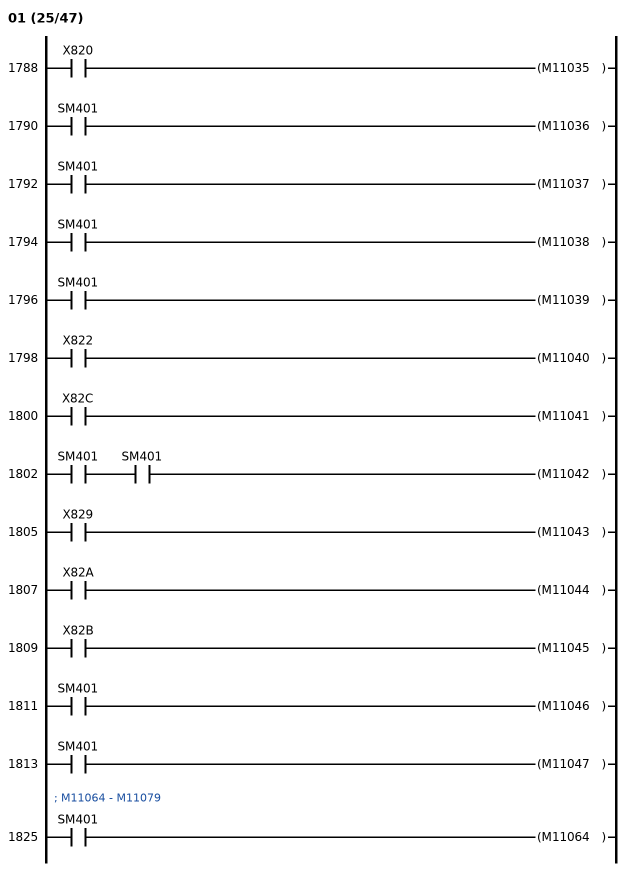
1788  LD      X820
      OUT     M11035
1790  LD      SM401
      OUT     M11036
1792  LD      SM401
      OUT     M11037
1794  LD      SM401
      OUT     M11038
1796  LD      SM401
      OUT     M11039
1798  LD      X822
      OUT     M11040
1800  LD      X82C
      OUT     M11041
1802  LD      SM401
      AND     SM401
      OUT     M11042
1805  LD      X829
      OUT     M11043
1807  LD      X82A
      OUT     M11044
1809  LD      X82B
      OUT     M11045
1811  LD      SM401
      OUT     M11046
1813  LD      SM401
      OUT     M11047
; M11064 - M11079
1825  LD      SM401
      OUT     M11064
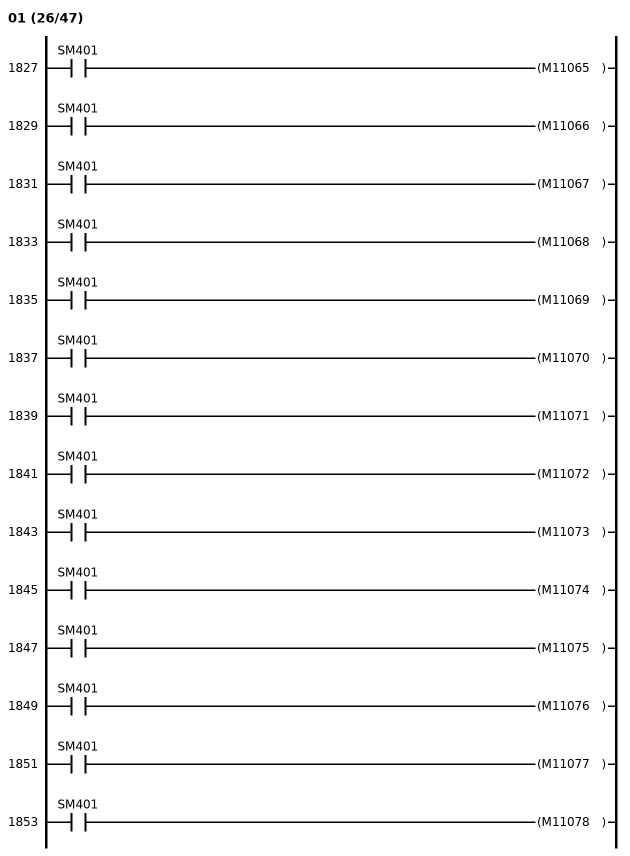
1827  LD      SM401
      OUT     M11065
1829  LD      SM401
      OUT     M11066
1831  LD      SM401
      OUT     M11067
1833  LD      SM401
      OUT     M11068
1835  LD      SM401
      OUT     M11069
1837  LD      SM401
      OUT     M11070
1839  LD      SM401
      OUT     M11071
1841  LD      SM401
      OUT     M11072
1843  LD      SM401
      OUT     M11073
1845  LD      SM401
      OUT     M11074
1847  LD      SM401
      OUT     M11075
1849  LD      SM401
      OUT     M11076
1851  LD      SM401
      OUT     M11077
1853  LD      SM401
      OUT     M11078
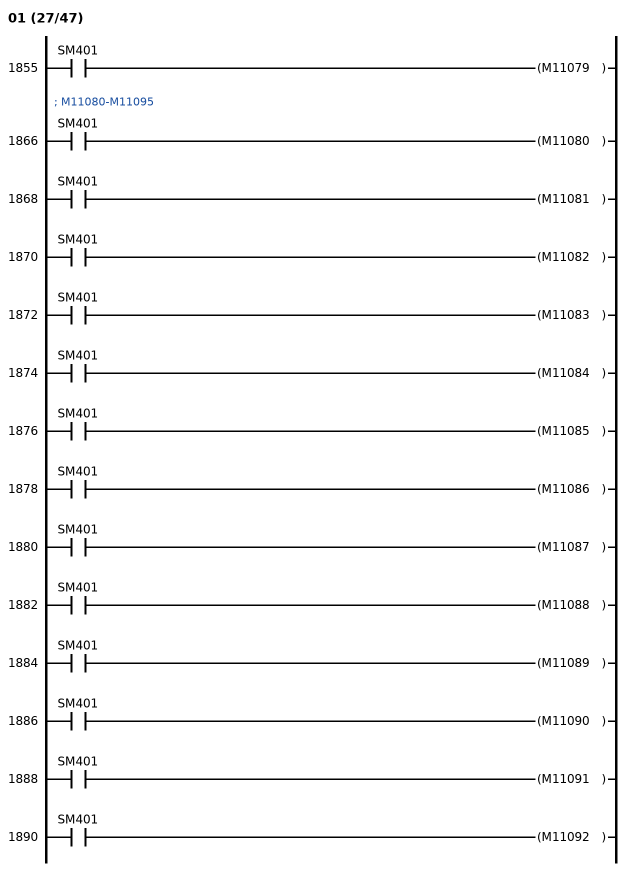
1855  LD      SM401
      OUT     M11079
; M11080-M11095
1866  LD      SM401
      OUT     M11080
1868  LD      SM401
      OUT     M11081
1870  LD      SM401
      OUT     M11082
1872  LD      SM401
      OUT     M11083
1874  LD      SM401
      OUT     M11084
1876  LD      SM401
      OUT     M11085
1878  LD      SM401
      OUT     M11086
1880  LD      SM401
      OUT     M11087
1882  LD      SM401
      OUT     M11088
1884  LD      SM401
      OUT     M11089
1886  LD      SM401
      OUT     M11090
1888  LD      SM401
      OUT     M11091
1890  LD      SM401
      OUT     M11092
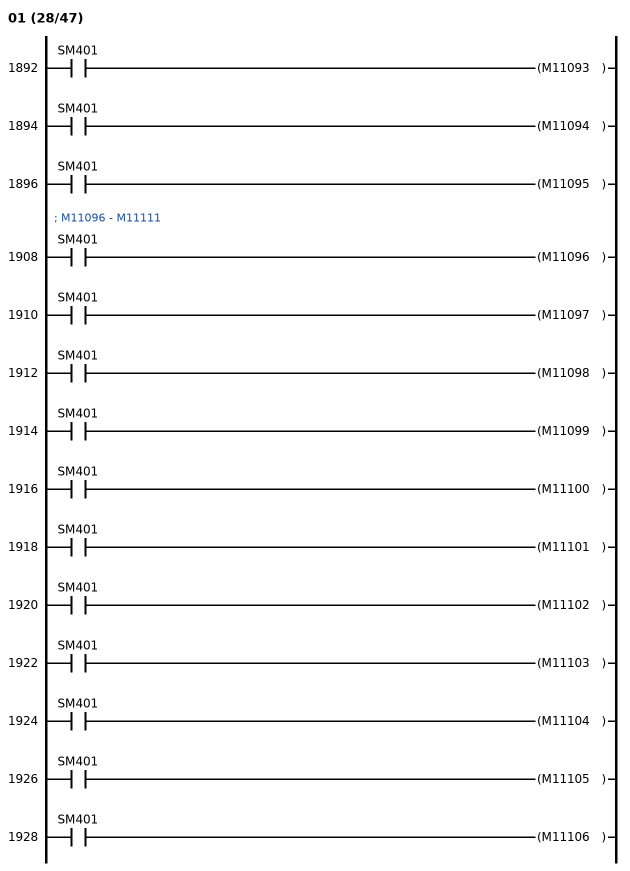
1892  LD      SM401
      OUT     M11093
1894  LD      SM401
      OUT     M11094
1896  LD      SM401
      OUT     M11095
; M11096 - M11111
1908  LD      SM401
      OUT     M11096
1910  LD      SM401
      OUT     M11097
1912  LD      SM401
      OUT     M11098
1914  LD      SM401
      OUT     M11099
1916  LD      SM401
      OUT     M11100
1918  LD      SM401
      OUT     M11101
1920  LD      SM401
      OUT     M11102
1922  LD      SM401
      OUT     M11103
1924  LD      SM401
      OUT     M11104
1926  LD      SM401
      OUT     M11105
1928  LD      SM401
      OUT     M11106
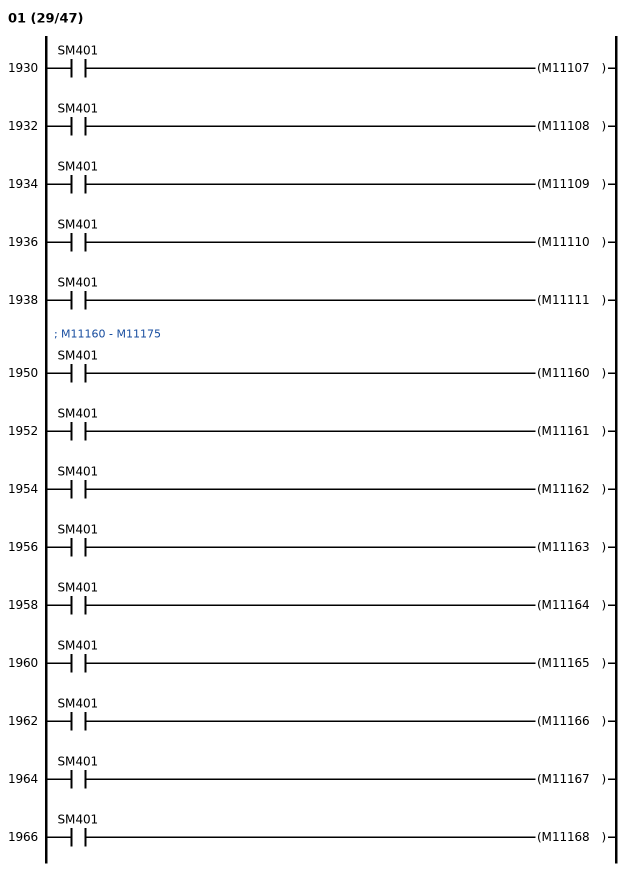
1930  LD      SM401
      OUT     M11107
1932  LD      SM401
      OUT     M11108
1934  LD      SM401
      OUT     M11109
1936  LD      SM401
      OUT     M11110
1938  LD      SM401
      OUT     M11111
; M11160 - M11175
1950  LD      SM401
      OUT     M11160
1952  LD      SM401
      OUT     M11161
1954  LD      SM401
      OUT     M11162
1956  LD      SM401
      OUT     M11163
1958  LD      SM401
      OUT     M11164
1960  LD      SM401
      OUT     M11165
1962  LD      SM401
      OUT     M11166
1964  LD      SM401
      OUT     M11167
1966  LD      SM401
      OUT     M11168
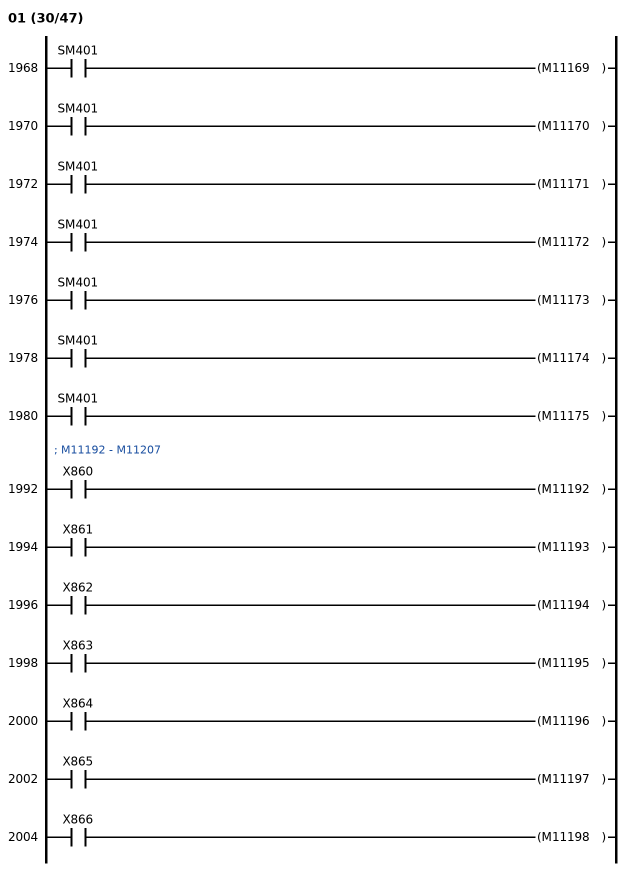
1968  LD      SM401
      OUT     M11169
1970  LD      SM401
      OUT     M11170
1972  LD      SM401
      OUT     M11171
1974  LD      SM401
      OUT     M11172
1976  LD      SM401
      OUT     M11173
1978  LD      SM401
      OUT     M11174
1980  LD      SM401
      OUT     M11175
; M11192 - M11207
1992  LD      X860
      OUT     M11192
1994  LD      X861
      OUT     M11193
1996  LD      X862
      OUT     M11194
1998  LD      X863
      OUT     M11195
2000  LD      X864
      OUT     M11196
2002  LD      X865
      OUT     M11197
2004  LD      X866
      OUT     M11198
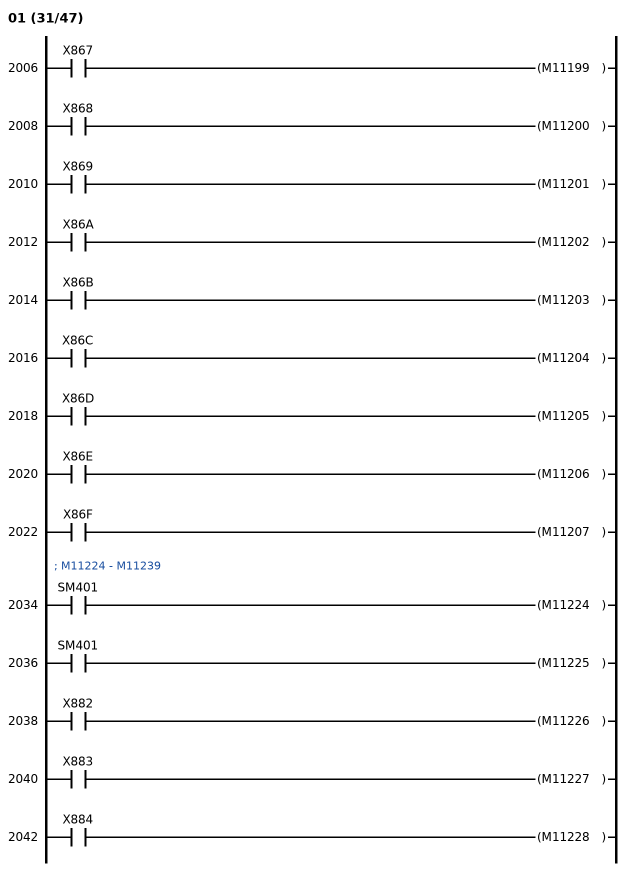
2006  LD      X867
      OUT     M11199
2008  LD      X868
      OUT     M11200
2010  LD      X869
      OUT     M11201
2012  LD      X86A
      OUT     M11202
2014  LD      X86B
      OUT     M11203
2016  LD      X86C
      OUT     M11204
2018  LD      X86D
      OUT     M11205
2020  LD      X86E
      OUT     M11206
2022  LD      X86F
      OUT     M11207
; M11224 - M11239
2034  LD      SM401
      OUT     M11224
2036  LD      SM401
      OUT     M11225
2038  LD      X882
      OUT     M11226
2040  LD      X883
      OUT     M11227
2042  LD      X884
      OUT     M11228
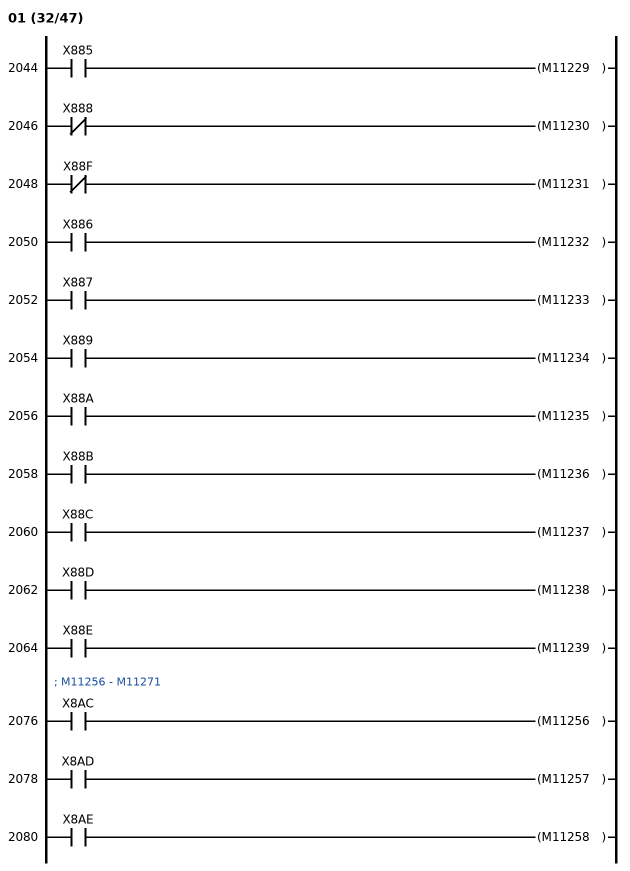
2044  LD      X885
      OUT     M11229
2046  LDI     X888
      OUT     M11230
2048  LDI     X88F
      OUT     M11231
2050  LD      X886
      OUT     M11232
2052  LD      X887
      OUT     M11233
2054  LD      X889
      OUT     M11234
2056  LD      X88A
      OUT     M11235
2058  LD      X88B
      OUT     M11236
2060  LD      X88C
      OUT     M11237
2062  LD      X88D
      OUT     M11238
2064  LD      X88E
      OUT     M11239
; M11256 - M11271
2076  LD      X8AC
      OUT     M11256
2078  LD      X8AD
      OUT     M11257
2080  LD      X8AE
      OUT     M11258
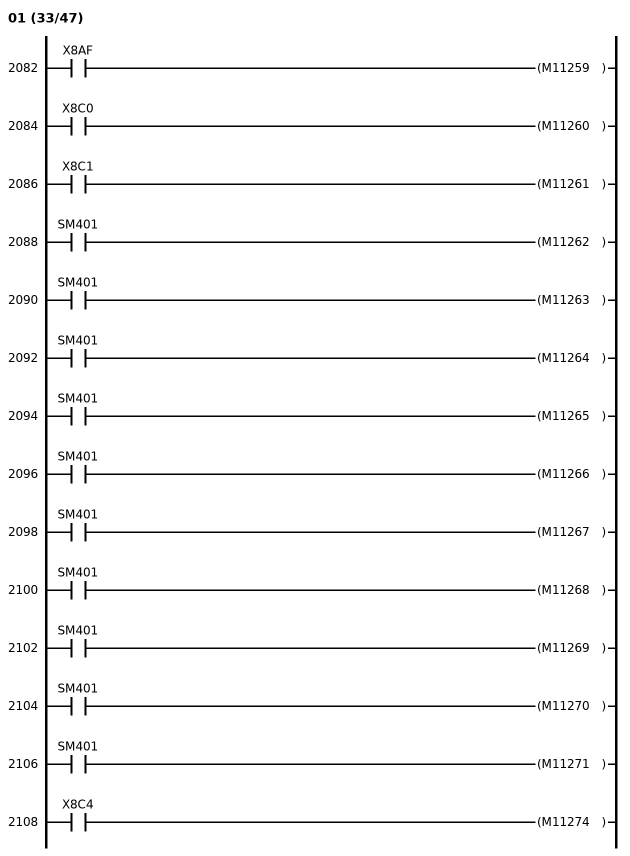
2082  LD      X8AF
      OUT     M11259
2084  LD      X8C0
      OUT     M11260
2086  LD      X8C1
      OUT     M11261
2088  LD      SM401
      OUT     M11262
2090  LD      SM401
      OUT     M11263
2092  LD      SM401
      OUT     M11264
2094  LD      SM401
      OUT     M11265
2096  LD      SM401
      OUT     M11266
2098  LD      SM401
      OUT     M11267
2100  LD      SM401
      OUT     M11268
2102  LD      SM401
      OUT     M11269
2104  LD      SM401
      OUT     M11270
2106  LD      SM401
      OUT     M11271
2108  LD      X8C4
      OUT     M11274
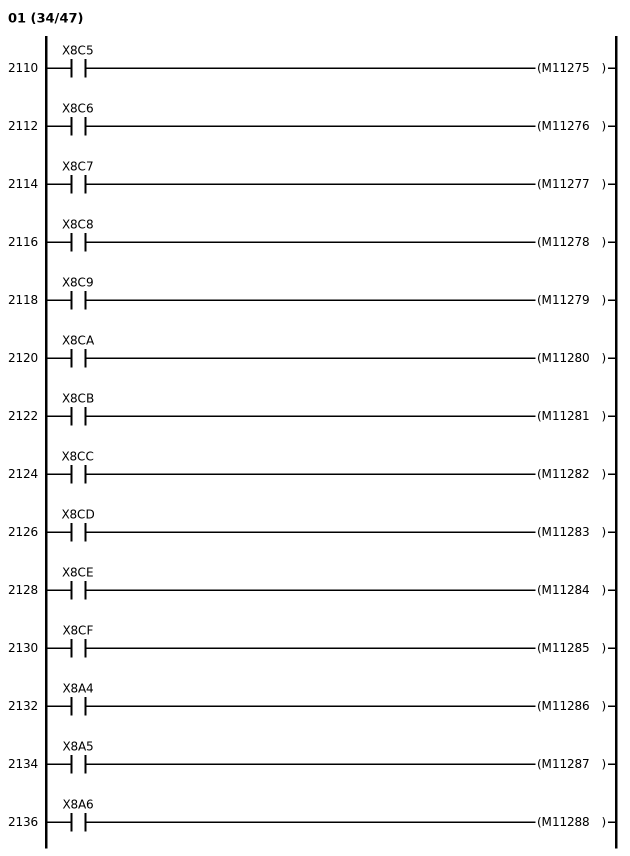
2110  LD      X8C5
      OUT     M11275
2112  LD      X8C6
      OUT     M11276
2114  LD      X8C7
      OUT     M11277
2116  LD      X8C8
      OUT     M11278
2118  LD      X8C9
      OUT     M11279
2120  LD      X8CA
      OUT     M11280
2122  LD      X8CB
      OUT     M11281
2124  LD      X8CC
      OUT     M11282
2126  LD      X8CD
      OUT     M11283
2128  LD      X8CE
      OUT     M11284
2130  LD      X8CF
      OUT     M11285
2132  LD      X8A4
      OUT     M11286
2134  LD      X8A5
      OUT     M11287
2136  LD      X8A6
      OUT     M11288
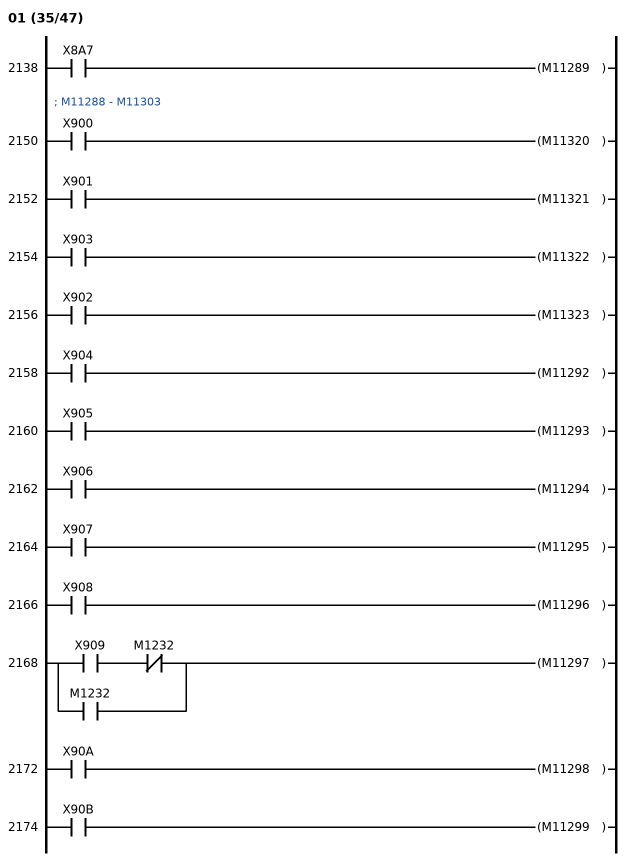
2138  LD      X8A7
      OUT     M11289
; M11288 - M11303
2150  LD      X900
      OUT     M11320
2152  LD      X901
      OUT     M11321
2154  LD      X903
      OUT     M11322
2156  LD      X902
      OUT     M11323
2158  LD      X904
      OUT     M11292
2160  LD      X905
      OUT     M11293
2162  LD      X906
      OUT     M11294
2164  LD      X907
      OUT     M11295
2166  LD      X908
      OUT     M11296
2168  LD      X909
      ANI     M1232
      OR      M1232
      OUT     M11297
2172  LD      X90A
      OUT     M11298
2174  LD      X90B
      OUT     M11299
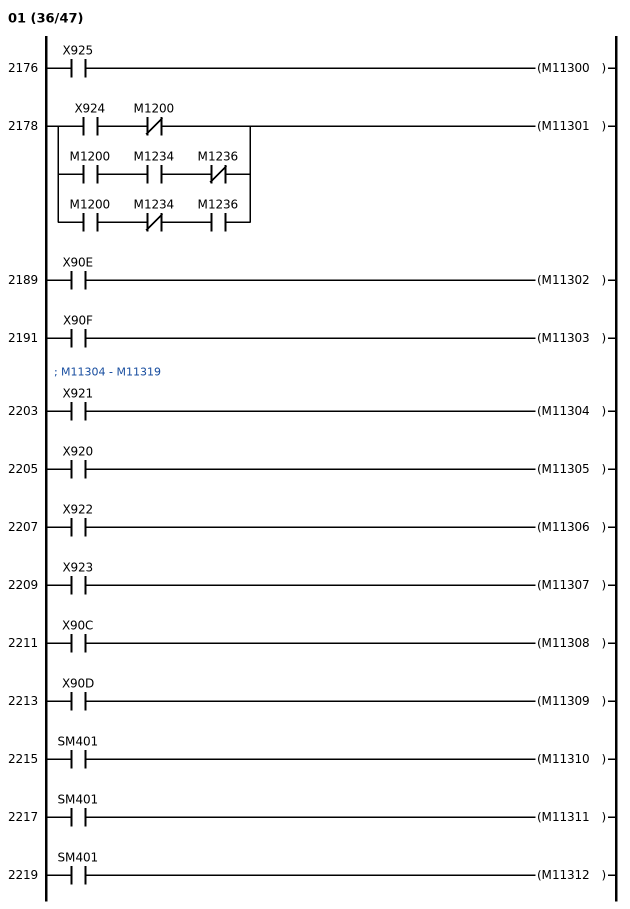
2176  LD      X925
      OUT     M11300
2178  LD      X924
      ANI     M1200
      LD      M1200
      AND     M1234
      ANI     M1236
      ORB
      LD      M1200
      ANI     M1234
      AND     M1236
      ORB
      OUT     M11301
2189  LD      X90E
      OUT     M11302
2191  LD      X90F
      OUT     M11303
; M11304 - M11319
2203  LD      X921
      OUT     M11304
2205  LD      X920
      OUT     M11305
2207  LD      X922
      OUT     M11306
2209  LD      X923
      OUT     M11307
2211  LD      X90C
      OUT     M11308
2213  LD      X90D
      OUT     M11309
2215  LD      SM401
      OUT     M11310
2217  LD      SM401
      OUT     M11311
2219  LD      SM401
      OUT     M11312
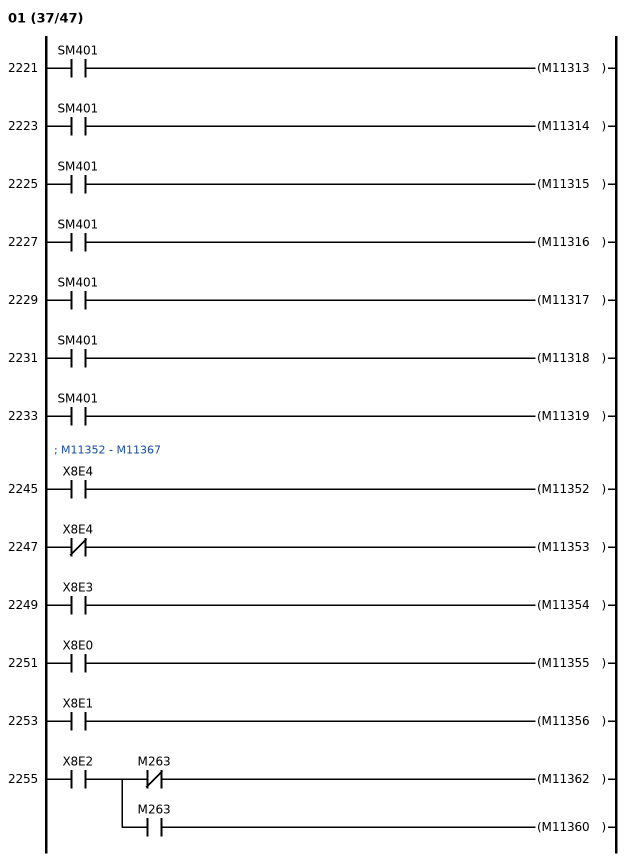
2221  LD      SM401
      OUT     M11313
2223  LD      SM401
      OUT     M11314
2225  LD      SM401
      OUT     M11315
2227  LD      SM401
      OUT     M11316
2229  LD      SM401
      OUT     M11317
2231  LD      SM401
      OUT     M11318
2233  LD      SM401
      OUT     M11319
; M11352 - M11367
2245  LD      X8E4
      OUT     M11352
2247  LDI     X8E4
      OUT     M11353
2249  LD      X8E3
      OUT     M11354
2251  LD      X8E0
      OUT     M11355
2253  LD      X8E1
      OUT     M11356
2255  LD      X8E2
      MPS
      ANI     M263
      OUT     M11362
      MPP
      AND     M263
      OUT     M11360
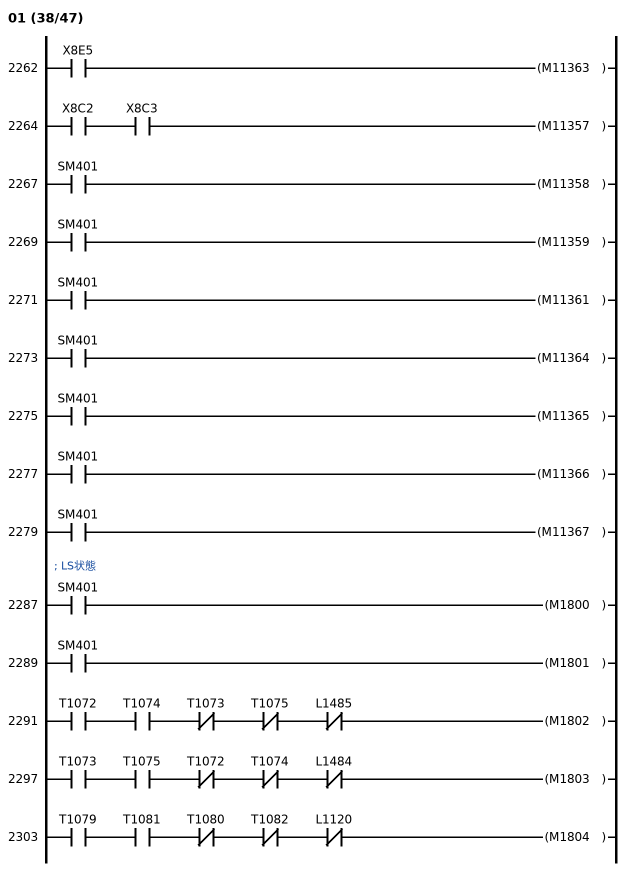
2262  LD      X8E5
      OUT     M11363
2264  LD      X8C2
      AND     X8C3
      OUT     M11357
2267  LD      SM401
      OUT     M11358
2269  LD      SM401
      OUT     M11359
2271  LD      SM401
      OUT     M11361
2273  LD      SM401
      OUT     M11364
2275  LD      SM401
      OUT     M11365
2277  LD      SM401
      OUT     M11366
2279  LD      SM401
      OUT     M11367
; LS状態
2287  LD      SM401
      OUT     M1800
2289  LD      SM401
      OUT     M1801
2291  LD      T1072
      AND     T1074
      ANI     T1073
      ANI     T1075
      ANI     L1485
      OUT     M1802
2297  LD      T1073
      AND     T1075
      ANI     T1072
      ANI     T1074
      ANI     L1484
      OUT     M1803
2303  LD      T1079
      AND     T1081
      ANI     T1080
      ANI     T1082
      ANI     L1120
      OUT     M1804
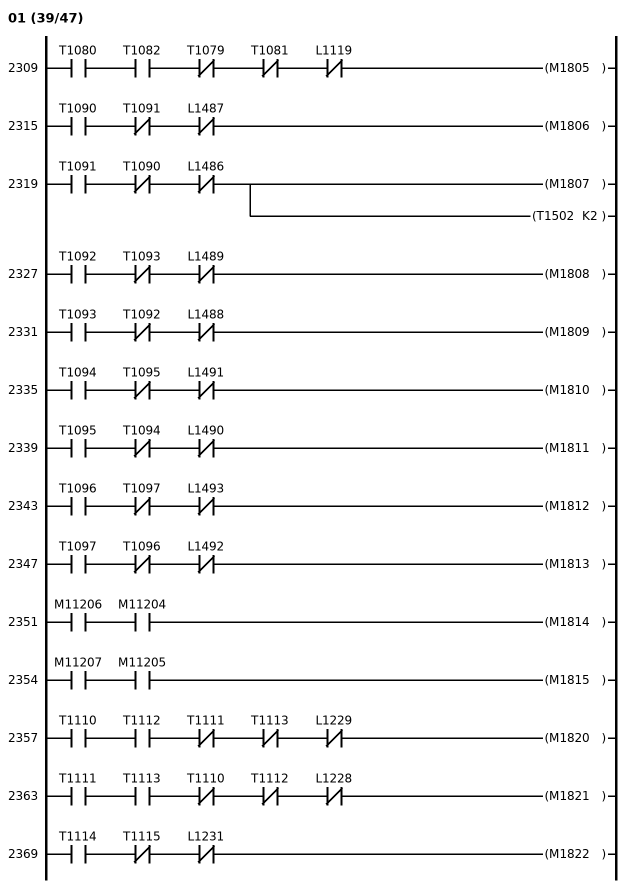
2309  LD      T1080
      AND     T1082
      ANI     T1079
      ANI     T1081
      ANI     L1119
      OUT     M1805
2315  LD      T1090
      ANI     T1091
      ANI     L1487
      OUT     M1806
2319  LD      T1091
      ANI     T1090
      ANI     L1486
      OUT     M1807
      OUT     T1502 K2
2327  LD      T1092
      ANI     T1093
      ANI     L1489
      OUT     M1808
2331  LD      T1093
      ANI     T1092
      ANI     L1488
      OUT     M1809
2335  LD      T1094
      ANI     T1095
      ANI     L1491
      OUT     M1810
2339  LD      T1095
      ANI     T1094
      ANI     L1490
      OUT     M1811
2343  LD      T1096
      ANI     T1097
      ANI     L1493
      OUT     M1812
2347  LD      T1097
      ANI     T1096
      ANI     L1492
      OUT     M1813
2351  LD      M11206
      AND     M11204
      OUT     M1814
2354  LD      M11207
      AND     M11205
      OUT     M1815
2357  LD      T1110
      AND     T1112
      ANI     T1111
      ANI     T1113
      ANI     L1229
      OUT     M1820
2363  LD      T1111
      AND     T1113
      ANI     T1110
      ANI     T1112
      ANI     L1228
      OUT     M1821
2369  LD      T1114
      ANI     T1115
      ANI     L1231
      OUT     M1822
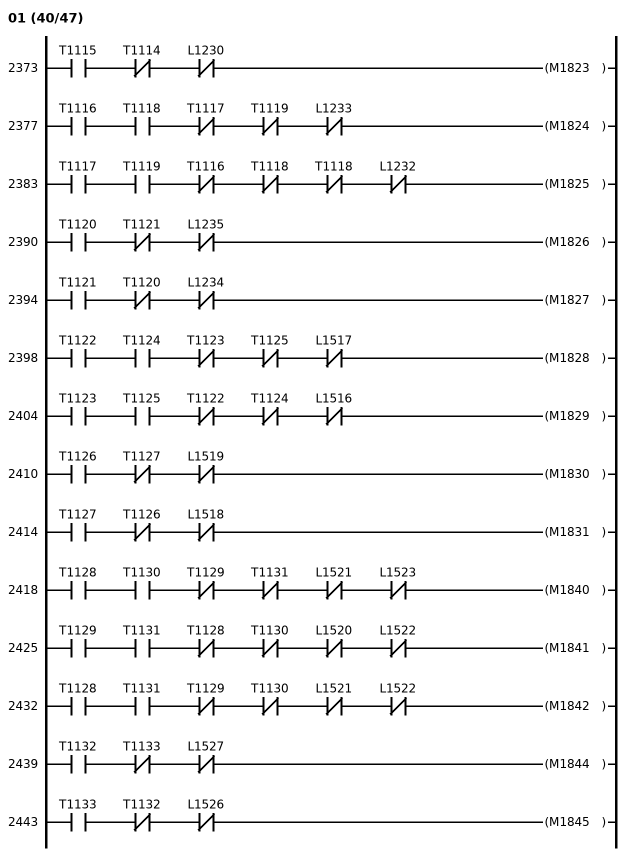
2373  LD      T1115
      ANI     T1114
      ANI     L1230
      OUT     M1823
2377  LD      T1116
      AND     T1118
      ANI     T1117
      ANI     T1119
      ANI     L1233
      OUT     M1824
2383  LD      T1117
      AND     T1119
      ANI     T1116
      ANI     T1118
      ANI     T1118
      ANI     L1232
      OUT     M1825
2390  LD      T1120
      ANI     T1121
      ANI     L1235
      OUT     M1826
2394  LD      T1121
      ANI     T1120
      ANI     L1234
      OUT     M1827
2398  LD      T1122
      AND     T1124
      ANI     T1123
      ANI     T1125
      ANI     L1517
      OUT     M1828
2404  LD      T1123
      AND     T1125
      ANI     T1122
      ANI     T1124
      ANI     L1516
      OUT     M1829
2410  LD      T1126
      ANI     T1127
      ANI     L1519
      OUT     M1830
2414  LD      T1127
      ANI     T1126
      ANI     L1518
      OUT     M1831
2418  LD      T1128
      AND     T1130
      ANI     T1129
      ANI     T1131
      ANI     L1521
      ANI     L1523
      OUT     M1840
2425  LD      T1129
      AND     T1131
      ANI     T1128
      ANI     T1130
      ANI     L1520
      ANI     L1522
      OUT     M1841
2432  LD      T1128
      AND     T1131
      ANI     T1129
      ANI     T1130
      ANI     L1521
      ANI     L1522
      OUT     M1842
2439  LD      T1132
      ANI     T1133
      ANI     L1527
      OUT     M1844
2443  LD      T1133
      ANI     T1132
      ANI     L1526
      OUT     M1845
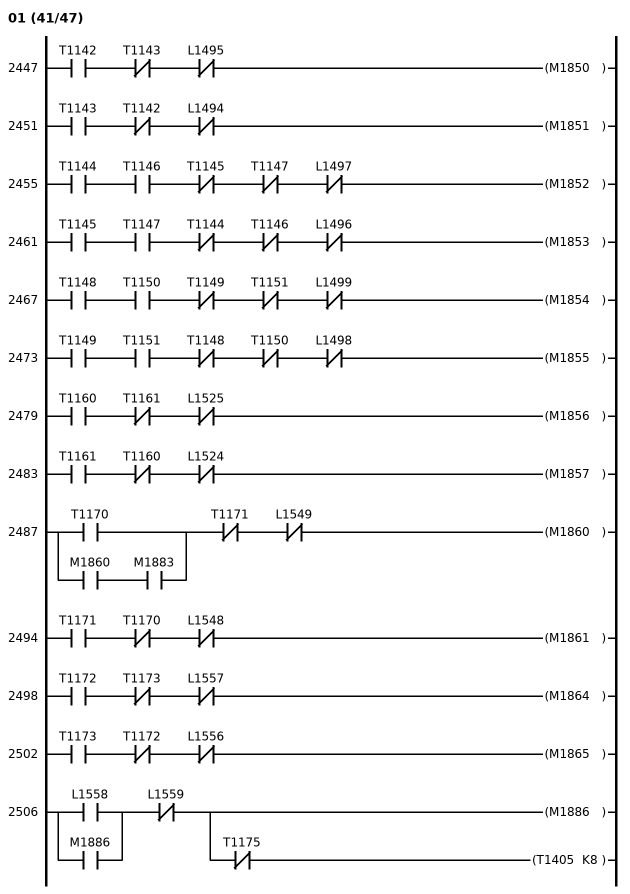
2447  LD      T1142
      ANI     T1143
      ANI     L1495
      OUT     M1850
2451  LD      T1143
      ANI     T1142
      ANI     L1494
      OUT     M1851
2455  LD      T1144
      AND     T1146
      ANI     T1145
      ANI     T1147
      ANI     L1497
      OUT     M1852
2461  LD      T1145
      AND     T1147
      ANI     T1144
      ANI     T1146
      ANI     L1496
      OUT     M1853
2467  LD      T1148
      AND     T1150
      ANI     T1149
      ANI     T1151
      ANI     L1499
      OUT     M1854
2473  LD      T1149
      AND     T1151
      ANI     T1148
      ANI     T1150
      ANI     L1498
      OUT     M1855
2479  LD      T1160
      ANI     T1161
      ANI     L1525
      OUT     M1856
2483  LD      T1161
      ANI     T1160
      ANI     L1524
      OUT     M1857
2487  LD      T1170
      LD      M1860
      AND     M1883
      ORB
      ANI     T1171
      ANI     L1549
      OUT     M1860
2494  LD      T1171
      ANI     T1170
      ANI     L1548
      OUT     M1861
2498  LD      T1172
      ANI     T1173
      ANI     L1557
      OUT     M1864
2502  LD      T1173
      ANI     T1172
      ANI     L1556
      OUT     M1865
2506  LD      L1558
      OR      M1886
      ANI     L1559
      OUT     M1886
      ANI     T1175
      OUT     T1405 K8
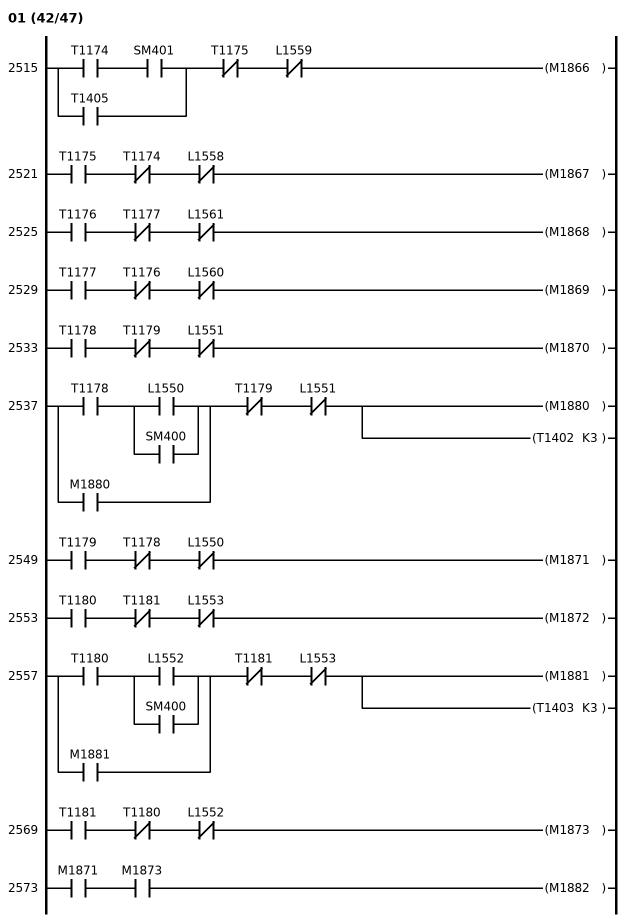
2515  LD      T1174
      AND     SM401
      OR      T1405
      ANI     T1175
      ANI     L1559
      OUT     M1866
2521  LD      T1175
      ANI     T1174
      ANI     L1558
      OUT     M1867
2525  LD      T1176
      ANI     T1177
      ANI     L1561
      OUT     M1868
2529  LD      T1177
      ANI     T1176
      ANI     L1560
      OUT     M1869
2533  LD      T1178
      ANI     T1179
      ANI     L1551
      OUT     M1870
2537  LD      T1178
      LD      L1550
      OR      SM400
      ANB
      OR      M1880
      ANI     T1179
      ANI     L1551
      OUT     M1880
      OUT     T1402 K3
2549  LD      T1179
      ANI     T1178
      ANI     L1550
      OUT     M1871
2553  LD      T1180
      ANI     T1181
      ANI     L1553
      OUT     M1872
2557  LD      T1180
      LD      L1552
      OR      SM400
      ANB
      OR      M1881
      ANI     T1181
      ANI     L1553
      OUT     M1881
      OUT     T1403 K3
2569  LD      T1181
      ANI     T1180
      ANI     L1552
      OUT     M1873
2573  LD      M1871
      AND     M1873
      OUT     M1882
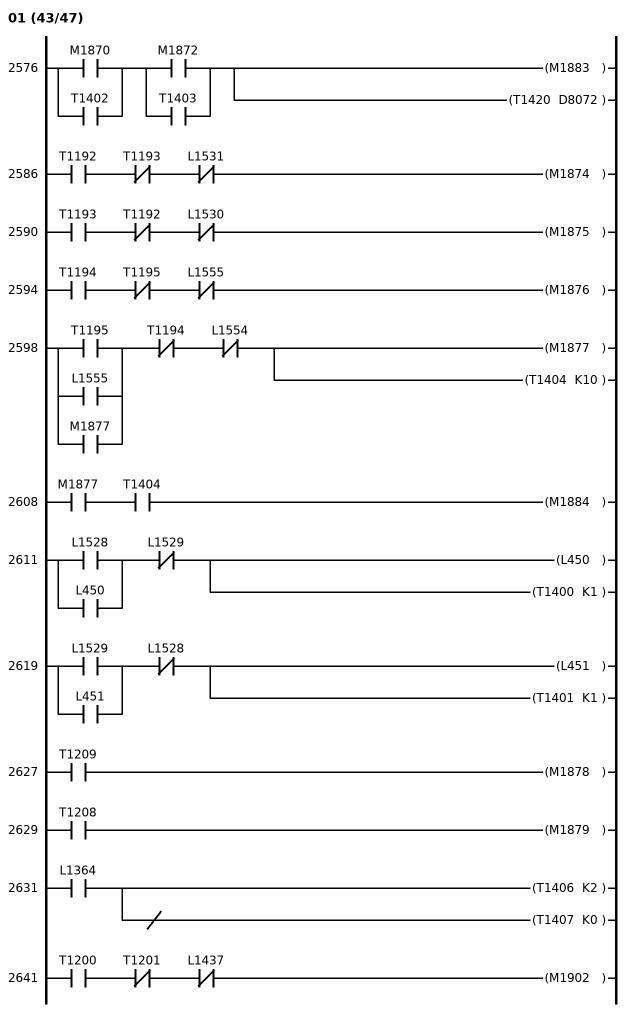
2576  LD      M1870
      OR      T1402
      LD      M1872
      OR      T1403
      ANB
      OUT     M1883
      OUT     T1420 D8072
2586  LD      T1192
      ANI     T1193
      ANI     L1531
      OUT     M1874
2590  LD      T1193
      ANI     T1192
      ANI     L1530
      OUT     M1875
2594  LD      T1194
      ANI     T1195
      ANI     L1555
      OUT     M1876
2598  LD      T1195
      OR      L1555
      OR      M1877
      ANI     T1194
      ANI     L1554
      OUT     M1877
      OUT     T1404 K10
2608  LD      M1877
      AND     T1404
      OUT     M1884
2611  LD      L1528
      OR      L450
      ANI     L1529
      OUT     L450
      OUT     T1400 K1
2619  LD      L1529
      OR      L451
      ANI     L1528
      OUT     L451
      OUT     T1401 K1
2627  LD      T1209
      OUT     M1878
2629  LD      T1208
      OUT     M1879
2631  LD      L1364
      OUT     T1406 K2
      INV
      OUT     T1407 K0
2641  LD      T1200
      ANI     T1201
      ANI     L1437
      OUT     M1902
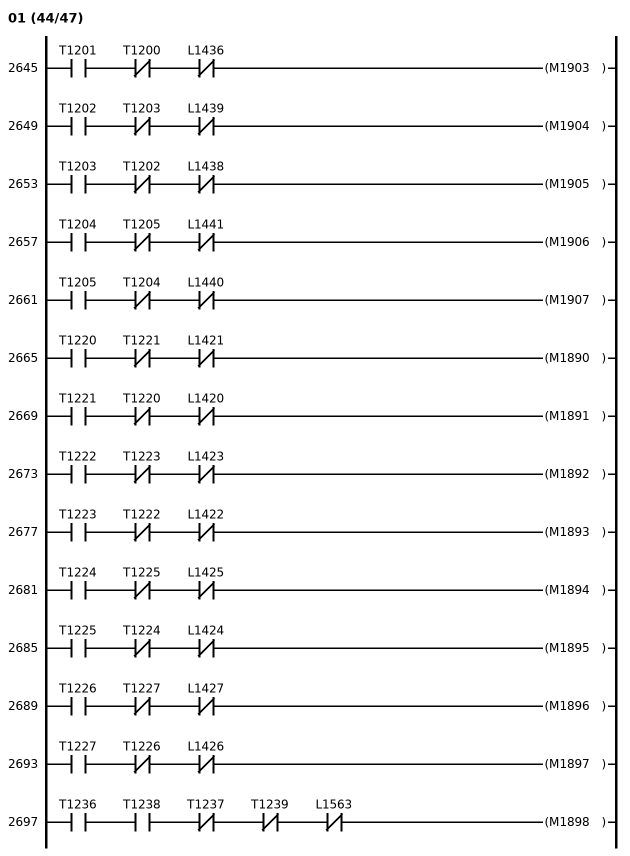
2645  LD      T1201
      ANI     T1200
      ANI     L1436
      OUT     M1903
2649  LD      T1202
      ANI     T1203
      ANI     L1439
      OUT     M1904
2653  LD      T1203
      ANI     T1202
      ANI     L1438
      OUT     M1905
2657  LD      T1204
      ANI     T1205
      ANI     L1441
      OUT     M1906
2661  LD      T1205
      ANI     T1204
      ANI     L1440
      OUT     M1907
2665  LD      T1220
      ANI     T1221
      ANI     L1421
      OUT     M1890
2669  LD      T1221
      ANI     T1220
      ANI     L1420
      OUT     M1891
2673  LD      T1222
      ANI     T1223
      ANI     L1423
      OUT     M1892
2677  LD      T1223
      ANI     T1222
      ANI     L1422
      OUT     M1893
2681  LD      T1224
      ANI     T1225
      ANI     L1425
      OUT     M1894
2685  LD      T1225
      ANI     T1224
      ANI     L1424
      OUT     M1895
2689  LD      T1226
      ANI     T1227
      ANI     L1427
      OUT     M1896
2693  LD      T1227
      ANI     T1226
      ANI     L1426
      OUT     M1897
2697  LD      T1236
      AND     T1238
      ANI     T1237
      ANI     T1239
      ANI     L1563
      OUT     M1898
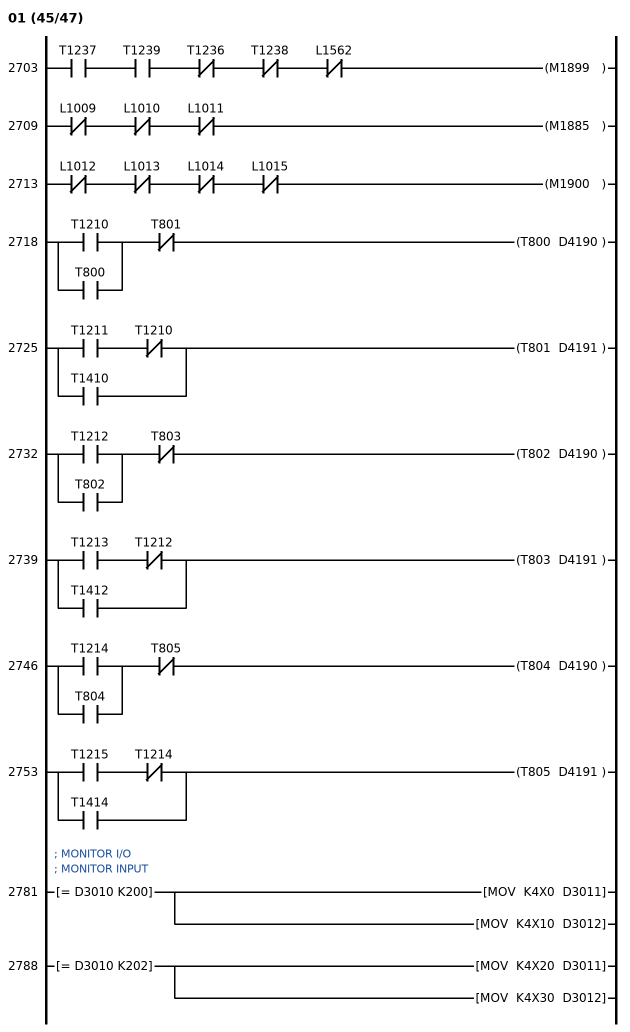
2703  LD      T1237
      AND     T1239
      ANI     T1236
      ANI     T1238
      ANI     L1562
      OUT     M1899
2709  LDI     L1009
      ANI     L1010
      ANI     L1011
      OUT     M1885
2713  LDI     L1012
      ANI     L1013
      ANI     L1014
      ANI     L1015
      OUT     M1900
2718  LD      T1210
      OR      T800
      ANI     T801
      OUT     T800 D4190
2725  LD      T1211
      ANI     T1210
      OR      T1410
      OUT     T801 D4191
2732  LD      T1212
      OR      T802
      ANI     T803
      OUT     T802 D4190
2739  LD      T1213
      ANI     T1212
      OR      T1412
      OUT     T803 D4191
2746  LD      T1214
      OR      T804
      ANI     T805
      OUT     T804 D4190
2753  LD      T1215
      ANI     T1214
      OR      T1414
      OUT     T805 D4191
; 
; MONITOR I/O
; 
; 
; MONITOR INPUT
; 
2781  LD=     D3010 K200
      MOV     K4X0 D3011
      MOV     K4X10 D3012
2788  LD=     D3010 K202
      MOV     K4X20 D3011
      MOV     K4X30 D3012
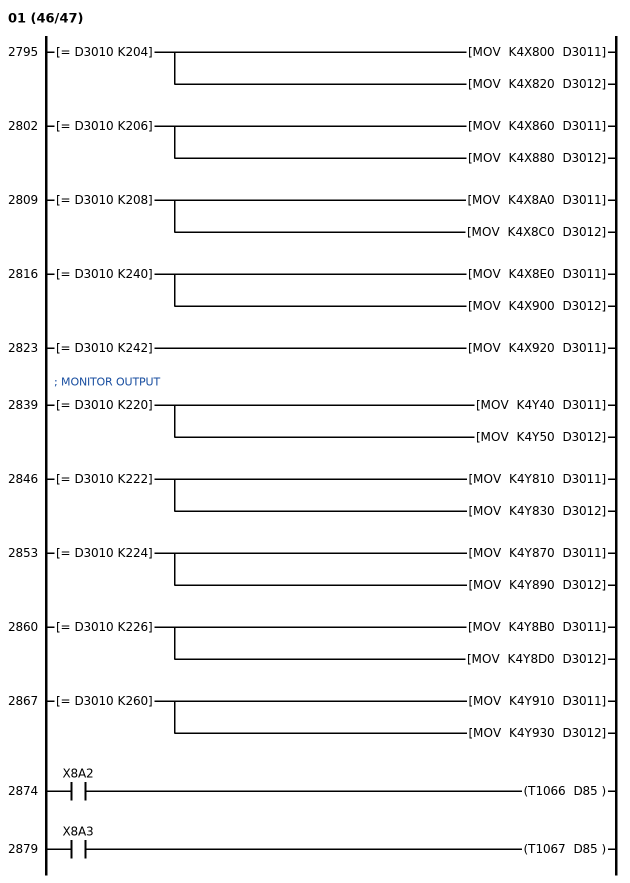
2795  LD=     D3010 K204
      MOV     K4X800 D3011
      MOV     K4X820 D3012
2802  LD=     D3010 K206
      MOV     K4X860 D3011
      MOV     K4X880 D3012
2809  LD=     D3010 K208
      MOV     K4X8A0 D3011
      MOV     K4X8C0 D3012
2816  LD=     D3010 K240
      MOV     K4X8E0 D3011
      MOV     K4X900 D3012
2823  LD=     D3010 K242
      MOV     K4X920 D3011
; 
; MONITOR OUTPUT
; 
2839  LD=     D3010 K220
      MOV     K4Y40 D3011
      MOV     K4Y50 D3012
2846  LD=     D3010 K222
      MOV     K4Y810 D3011
      MOV     K4Y830 D3012
2853  LD=     D3010 K224
      MOV     K4Y870 D3011
      MOV     K4Y890 D3012
2860  LD=     D3010 K226
      MOV     K4Y8B0 D3011
      MOV     K4Y8D0 D3012
2867  LD=     D3010 K260
      MOV     K4Y910 D3011
      MOV     K4Y930 D3012
2874  LD      X8A2
      OUT     T1066 D85
2879  LD      X8A3
      OUT     T1067 D85
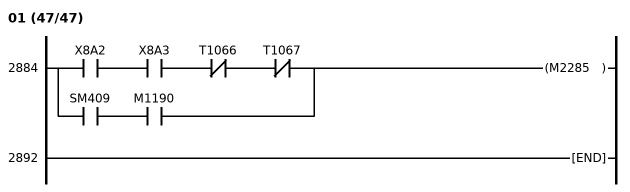
2884  LD      X8A2
      AND     X8A3
      ANI     T1066
      ANI     T1067
      LD      SM409
      AND     M1190
      ORB
      OUT     M2285
2892  END
END_PROGRAM

PROGRAM 10
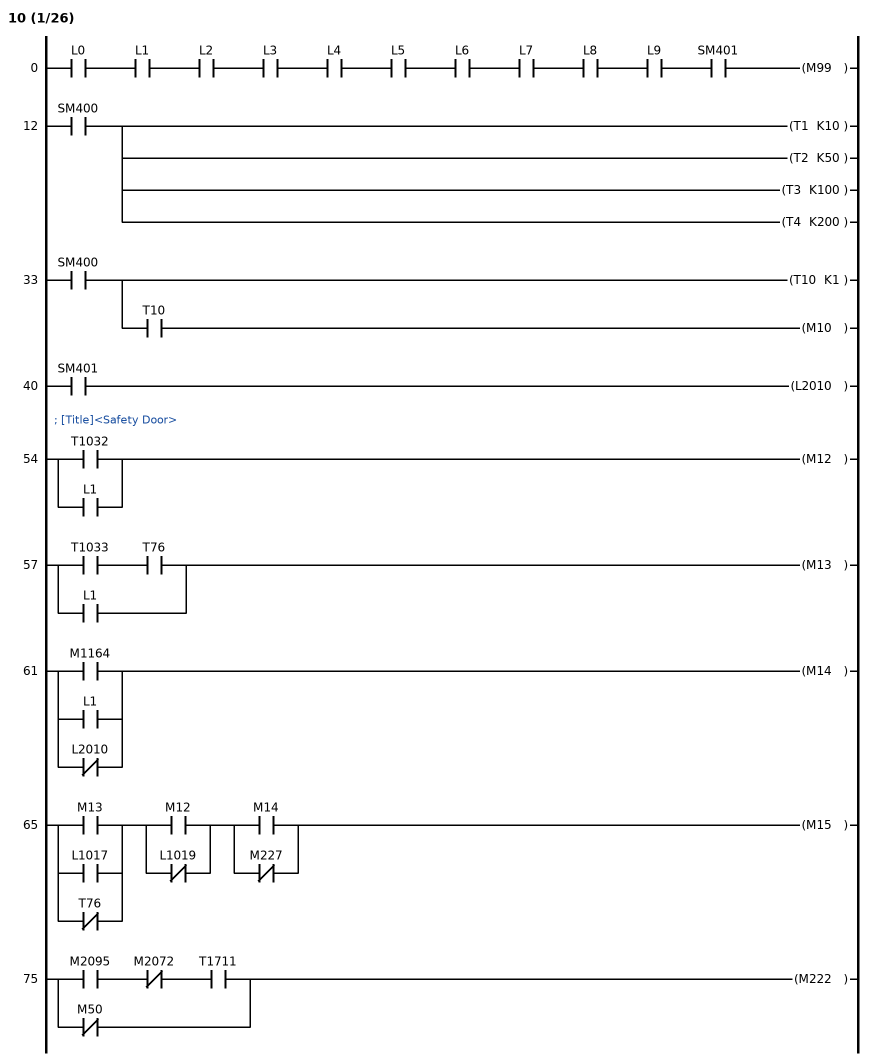
0     LD      L0
      AND     L1
      AND     L2
      AND     L3
      AND     L4
      AND     L5
      AND     L6
      AND     L7
      AND     L8
      AND     L9
      AND     SM401
      OUT     M99
12    LD      SM400
      OUT     T1 K10
      OUT     T2 K50
      OUT     T3 K100
      OUT     T4 K200
; 
; 
; 
33    LD      SM400
      OUT     T10 K1
      AND     T10
      OUT     M10
40    LD      SM401
      OUT     L2010
; [Title]<Safety Door>
54    LD      T1032
      OR      L1
      OUT     M12
57    LD      T1033
      AND     T76
      OR      L1
      OUT     M13
61    LD      M1164
      OR      L1
      ORI     L2010
      OUT     M14
65    LD      M13
      OR      L1017
      ORI     T76
      LD      M12
      ORI     L1019
      ANB
      LD      M14
      ORI     M227
      ANB
      OUT     M15
75    LD      M2095
      ANI     M2072
      AND     T1711
      ORI     M50
      OUT     M222
